// TIA Portal V19 export
DATA_BLOCK "Alarms"   // DB59
// stored: Access Published, MemoryReserve 100, Namespace Unit3
   VAR
      unitAlarms { ExternalWritable := 'False'} : "LAF_typeAlarms";
      emAlarms { ExternalWritable := 'False'} : Array[0.._.Unit3_NO_OF_EMs] of "LAF_typeAlarms";
      errorNoReaction { ExternalWritable := 'False'} : Array[0..9] of Bool;   // Error without further impact / Error ohne weitere Auswirkungen
      errorAbort { ExternalWritable := 'False'} : Array[0..9] of Bool;   // Error which aborts the whole Unit / Error der ein abort in der Unit auslöst
      errorStop { ExternalWritable := 'False'} : Array[0..9] of Bool;   // Error which stops the whole Unit / Error der ein stop in der Unit auslöst
      warningNoReaction { ExternalWritable := 'False'} : Array[0..9] of Bool;   // Warning which could lead to a error / Warnung die zu einem Error führen kann
      warningHold { ExternalWritable := 'False'} : Array[0..9] of Bool;   // Warning which holds the whole Unit / Warnung die ein hold in der Unit auslöst
      warningSuspend { ExternalWritable := 'False'} : Array[0..9] of Bool;   // Warning which suspends the whole Unit / Warnung die ein suspend in der Unit auslöst
      information { ExternalWritable := 'False'} : Array[0..9] of Bool;   // Informations of the EM / Information der Unit
      criteriaAnalysis { ExternalWritable := 'False'} : Array[0..9] of Bool;   // CriteriaAnalysis of the EM / Kriterienanalyse der Unit
   END_VAR
BEGIN
   // errorNoReaction[0] : Error in subordinated Modules / Error in untergelagertem Modul
   // errorStop[0] : Error which stops the whole Unit / Error der ein stop in der Unit auslöst
   // warningNoReaction[0] : Warning in subordinated Modules / Warnung in untergelagertem Modul
   // warningHold[0] : Warning which holds the whole Unit / Warnung die ein hold in der Unit auslöst
   // warningSuspend[0] : Warning which suspends the whole Unit / Warnung die ein suspend in der Unit auslöst
   information[0] := false;   // Information in subordinated Modules / Information in untergelagertem Modul
   // criteriaAnalysis[0] : CriteriaAnalysis of the EM / Safety Acknowledge wird angefordert
END_DATA_BLOCK
